FUNCTION F_PB_GetTransportData : ST_TransportData
(**************************************************************************************
 * 	Application		:	BoxControl Framework
 *	Revision		:	$Revision:  $
 *	Revision date	:	$Date: $
 *	Last changed by	:	$Author: q8sheds $
 *	URL				:	$URL: $
 *
 *	Purpose			:	return Transport data
 *
 * ------------------------------------------------------------------------------------
 *	Copyright Swisslog [IP AG], Switzerland. All rights reserved.
 * 
 * ------------------------------------------------------------------------------------
 *	
 * 	Revision History: 
 *
 * 	VERSION			DATE			INITIALS			DESCRIPTION
 *	0.1				01.01.2001		swl					Example
 *
 **************************************************************************************)
VAR_INPUT
	eFunctionNumber		: E_FunctionNumber; // Function number
	ZoneNumber			: INT; // Zone number
END_VAR



VAR
	FunctionBase: INT;
END_VAR


//init default data
F_PB_GetTransportData.eFunctionNumber := E_FunctionNumber.F_BEGIN_FUNCTION;
F_PB_GetTransportData.ZoneNumber:=0;
F_PB_GetTransportData.rTransportControlData REF= PBTransportCtrl.pbTransportControlDataEmpty;
F_PB_GetTransportData.rSettings REF= PBTransportCtrl.pbZoneSettingsEmpty;


// Check if function number is valid
IF eFunctionNumber > E_FunctionNumber.F_BEGIN_FUNCTION AND
   eFunctionNumber < E_FunctionNumber.F_END_FUNCTION AND
   ZoneNumber > 0 AND ZoneNumber <= NUMBER_OF_ZONES_PER_FUNCTION THEN
  
	// Check reference is valid
	IF __ISVALIDREF(FunctionRegistry[eFunctionNumber].Zone[ZoneNumber].refZoneData) THEN
   		// Set transport data
   		//F_PB_GetTransportControlDataRef REF= FunctionRegistry[eFunctionNumber].Zone[ZoneNumber].refZoneData.TransportControlData;
		F_PB_GetTransportData.eFunctionNumber := eFunctionNumber;
		F_PB_GetTransportData.ZoneNumber := ZoneNumber;
		F_PB_GetTransportData.rSettings REF= FunctionRegistry[eFunctionNumber].rSettingsFunction.Zone[ZoneNumber];
		F_PB_GetTransportData.rTransportControlData REF= FunctionRegistry[eFunctionNumber].Zone[ZoneNumber].refZoneData.TransportControlData;				
	END_IF
END_IF

END_FUNCTION

(* stored: Version 1.1.0.1, ProductVersion 3.1.4022.12
   POU F_PB_GetTransportData: Id {bfa77049-55f9-4131-8a55-0529d7952f65}, SpecialFunc None *)
